(* Schneider Machine Expert - Basic project Grafcet prgram, file version 2.7.0.0 *)
(* ProjectInformations: Name=Nuevo proyecto *)

HARDWARE
  Cpu 0: TM221M16R/G
  ModuleExtensionObject 0: TM3DI16K
  EthernetConfiguration: NetworkName=M221, IpAllocationMode=FixedAddress, IpAddress=0.0.0.0, SubnetMask=0.0.0.0
  SerialLineConfiguration: Baud=Baud19200, Parity=ParityEven, DataBits=DataBits8, StopBits=StopBits1, PhysicalMedium=PhysicalMediumRs485, TransmissionMode=TransmissionModeModbusRtu, SlaveId=1, Addressing=SlaveAddressing
  MastTask: UsePeriodScanMode=false, PeriodScan=100
  FastTask: Period=255
  CpuBehavior: StartingMode=StartAsPreviousState, AutoSaveRamOnEeprom=true, WatchdogPeriod=250

SYMBOLS  (address, symbol, comment, settings)
  %M0         "Item at entry"
  %M1         "Item at exit"
  %M2         "Moving X"
  %M3         "Moving Z"
  %M4         "Item detected"
  %M5         "Lids center (busy)"
  %M11        "Entry conveyor"
  %M12        "Exit conveyor"
  %M13        "Move X"
  %M14        "Move Z"
  %M15        "Grab"
  %TM0        "Temporizador estado 3"  [Preset=1, Base=OneSecond]
  %TM1        "Temporizador estado 4"  [Preset=1, Base=OneSecond]
  %TM2        "Temporizador estado 7"  [Preset=1, Base=OneSecond]
  %TM3        "Aux"  [Type=TOF, Preset=12, Base=OneSecond]

GRAFCET Grafcet POU
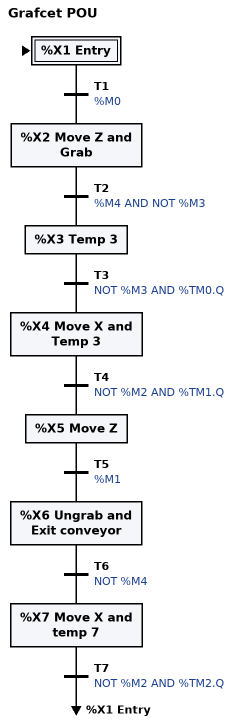
  INITIAL_STEP %X1  (* Entry *)
  STEP %X2  (* Move Z and Grab *)
  STEP %X3  (* Temp 3 *)
  STEP %X4  (* Move X and Temp 3 *)
  STEP %X5  (* Move Z *)
  STEP %X6  (* Ungrab and Exit conveyor *)
  STEP %X7  (* Move X and temp 7 *)
  TRANSITION T1 FROM %X1 TO %X2 := %M0;
  TRANSITION T2 FROM %X2 TO %X3 := %M4 AND NOT %M3;
  TRANSITION T3 FROM %X3 TO %X4 := NOT %M3 AND %TM0.Q;
  TRANSITION T4 FROM %X4 TO %X5 := NOT %M2 AND %TM1.Q;
  TRANSITION T5 FROM %X5 TO %X6 := %M1;
  TRANSITION T6 FROM %X6 TO %X7 := NOT %M4;
  TRANSITION T7 FROM %X7 TO %X1 := NOT %M2 AND %TM2.Q;

TRANSITION T1 (%X1 -> %X2) 
  (* SectionNumber=0 *)

// Rung 0: Tr1
  LD %M0
  ENDT
  // as ST:
  //   TRANSITION := %M0;

TRANSITION T2 (%X2 -> %X3) 
  (* SectionNumber=0 *)

// Rung 1: Tr2
  LD %M4
  ANDN %M3
  ENDT
  // as ST:
  //   TRANSITION := %M4 AND NOT %M3;

TRANSITION T3 (%X3 -> %X4) 
  (* SectionNumber=0 *)

// Rung 2: Tr3
  LDN %M3
  AND %TM0.Q
  ENDT
  // as ST:
  //   TRANSITION := NOT %M3 AND %TM0.Q;

TRANSITION T4 (%X4 -> %X5) 
  (* SectionNumber=0 *)

// Rung 3: Tr4
  LDN %M2
  AND %TM1.Q
  ENDT
  // as ST:
  //   TRANSITION := NOT %M2 AND %TM1.Q;

TRANSITION T5 (%X5 -> %X6) 
  (* SectionNumber=0 *)

// Rung 4: Tr5
  LD %M1
  ENDT
  // as ST:
  //   TRANSITION := %M1;

TRANSITION T6 (%X6 -> %X7) 
  (* SectionNumber=0 *)

// Rung 5: Tr6
  LDN %M4
  ENDT
  // as ST:
  //   TRANSITION := NOT %M4;

TRANSITION T7 (%X7 -> %X1) 
  (* SectionNumber=0 *)

// Rung 6: Tr7
  LDN %M2
  AND %TM2.Q
  ENDT
  // as ST:
  //   TRANSITION := NOT %M2 AND %TM2.Q;

POU Acciones
  (* SectionNumber=9 *)

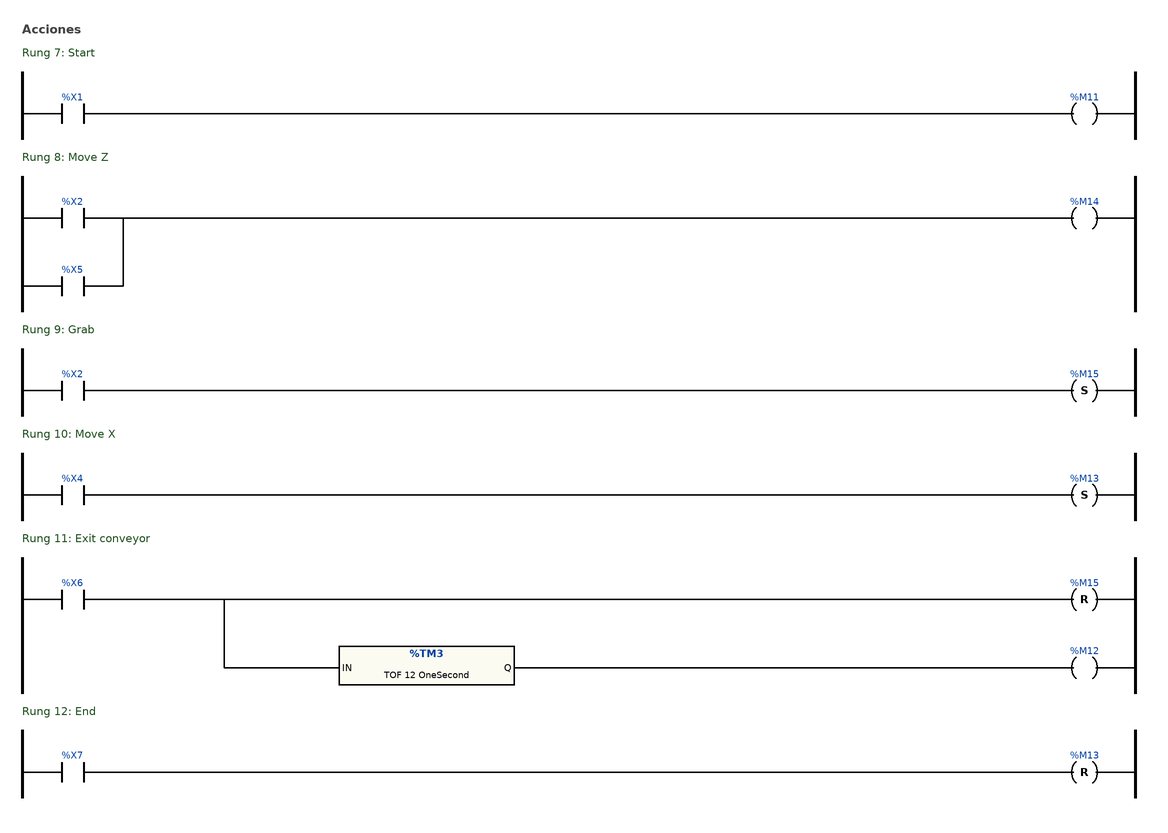

// Rung 7: Start
  LD %X1
  ST %M11
  // as ST:
  //   %M11 := %X1;

// Rung 8: Move Z
  LD %X2
  OR %X5
  ST %M14
  // as ST:
  //   %M14 := %X2 OR %X5;

// Rung 9: Grab
  LD %X2
  S %M15
  // as ST:
  //   IF %X2 THEN %M15 := TRUE; END_IF;

// Rung 10: Move X
  LD %X4
  S %M13
  // as ST:
  //   IF %X4 THEN %M13 := TRUE; END_IF;

// Rung 11: Exit conveyor
  LD 1
  MULTIFB
  LD 1
  AND %X6
  ST %MW2009:X0
  LD %MW2009:X0
  R %M15
  BLK %TM3
  LD %MW2009:X0
  IN
  OUT_BLK
  LD Q
  ST %M12
  END_BLK
  MULTIFB
  // as ST:
  //   IF %X6 THEN %M15 := FALSE; END_IF;
  //   %TM3(IN := %X6);
  //   %M12 := %TM3.Q;

// Rung 12: End
  LD %X7
  R %M13
  // as ST:
  //   IF %X7 THEN %M13 := FALSE; END_IF;

POU Temporizadores y contadores
  (* SectionNumber=10 *)

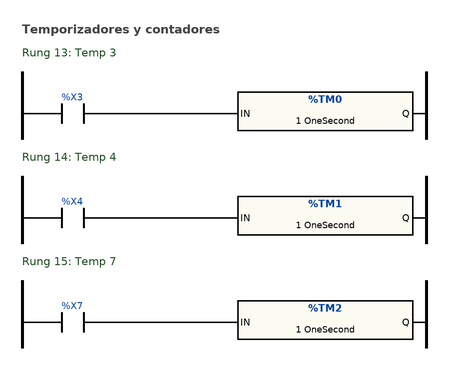

// Rung 13: Temp 3
  BLK %TM0
  LD %X3
  IN
  END_BLK
  // as ST:
  //   %TM0(IN := %X3);

// Rung 14: Temp 4
  BLK %TM1
  LD %X4
  IN
  END_BLK
  // as ST:
  //   %TM1(IN := %X4);

// Rung 15: Temp 7
  BLK %TM2
  LD %X7
  IN
  END_BLK
  // as ST:
  //   %TM2(IN := %X7);
